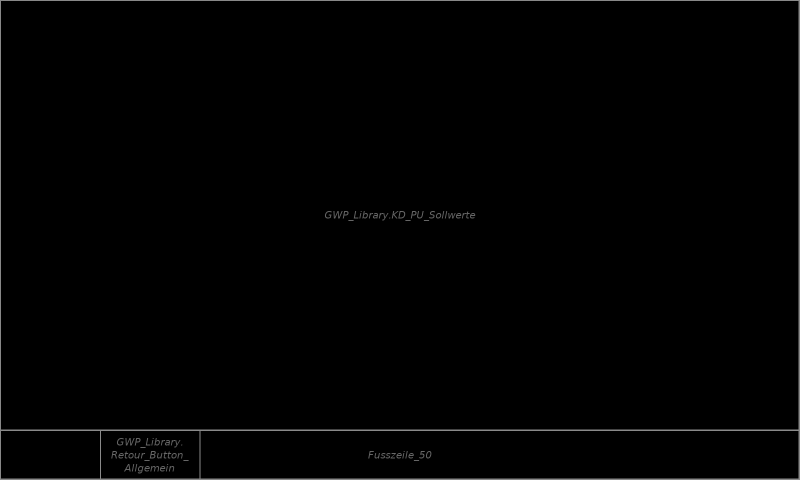
VISUALIZATION KD_PU_Sollwerte  // 800x480
    Frame (0,0 800x430)
        shows GWP_Library.KD_PU_Sollwerte(FB_KD := Main.KD_0)
    Frame (0,430 800x50)
        shows Fusszeile_50()
    Frame (100,430 100x50)
        shows GWP_Library.Retour_Button_Allgemein()
END_VISUALIZATION

(* stored: Version 1.1.0.1, ProductVersion 3.1.4022.6
   Visu KD_PU_Sollwerte: Id {ecfcd9b1-48db-44d3-9c2c-844b25000e32} *)
